FUNCTION_BLOCK SafetyOkVisitor IMPLEMENTS I_ComponentVisitor
VAR
	{attribute 'hide'}
	_OK				: BOOL;
	SafetyComponent : I_SafetyBase;
	ErrorComponent	: I_Component;
END_VAR

METHOD Check
VAR_INPUT
	Components : I_ComponentCollection;
END_VAR
_OK := TRUE;
Components.Accept(THIS^);
END_METHOD

{attribute 'monitoring' := 'call'}
PROPERTY OK : BOOL
GET
OK := _OK;
END_GET
END_PROPERTY

METHOD VisitComponent
VAR_INPUT
	Component : I_Component;
END_VAR
IF __QUERYINTERFACE(Component, SafetyComponent) THEN
	IF NOT SafetyComponent.OK THEN
		ErrorComponent := Component;
		_OK			   := FALSE;
	END_IF
END_IF
END_METHOD

END_FUNCTION_BLOCK

(* stored: Version 1.1.0.1, ProductVersion 3.1.4026.18
   POU SafetyOkVisitor: Id {fb66a7e7-6422-4f74-a738-89af8bbbdcdb}, SpecialFunc None
   Method Check: Id {5c980e43-1276-4f1c-a8c8-9c7272ab30b3}
   Property OK: Id {1340a3f4-d616-4d71-ad45-b35527c94ce3}
   Get Get: Id {93e58e58-de31-4f90-b314-89893d0ca755}
   Method VisitComponent: Id {162ccdde-fdb2-4cb6-91bd-31788e7ad38b} *)
